TYPE ST_REQUEST_LINE :
STRUCT
	eMethod 	: E_METHOD;
	sURI 		: T_MaxString;
	sProtocol 	: T_MaxString;
END_STRUCT
END_TYPE

(* stored: Version 1.1.0.1, ProductVersion 3.1.4024.4
   DUT ST_REQUEST_LINE: Id {0a605d18-87c3-423a-9448-4dc14424ea79} *)
